(*
:Description: User-facing FB for capturing oversampled metric values and pushing
to tc-otel as compact batched frames.

Lifecycle pattern: declare one FB_Metrics per logical metric, ``Init`` it once
in first cycle, then call ``Observe`` with the value of any IEC scalar (or
STRING / WSTRING) you want to track. The FB:

* Locks the IEC type class on the very first ``Observe`` and rejects later
  calls of a different class — no aggregator-strategy switching mid-flight.
* Optionally rate-limits sampling (``SetSampleIntervalMs``) so a value that
  changes faster than the configured interval is sampled at most once per
  interval. Default 0 = no rate limit (every change is sampled).
* Optionally suppresses redundant samples (``SetChangeDetect``, default TRUE)
  via byte-wise comparison against the last sampled value.
* Buffers samples in an append-only body buffer (8 KB default). On overflow
  the per-frame ``flags.bit1 = ring_overflowed`` is set and additional
  samples are dropped until the next flush.
* Flushes the buffer at the configured push interval (``SetPushIntervalMs``,
  default 1000 ms). Flush also fires from ``Call()`` so users who call
  ``Observe`` only on demand still get punctual pushes.

Each frame carries header + (optional trace context) + name + unit + body.
The body is just ``sample_count * sample_size`` raw bytes — no per-sample
type/length, the receiver knows the layout from the header's ``body_schema``.

Numerics (all signed/unsigned int + REAL + LREAL) widen to LREAL (8 B). BOOL
is one byte. STRING/WSTRING are zero-padded to a per-instance fixed size
configured in ``Init``. Discrete byte-types (BYTE/WORD/DWORD/LWORD/ENUM)
are shipped raw at their native size.

**Example**

.. code-block:: pascal

    VAR
        fbMotorTemp : FB_Metrics;
    END_VAR

    IF _TaskInfo[GETCURTASKINDEXEX()].FirstCycle THEN
        fbMotorTemp.Init('motor.temperature', 'celsius');
        fbMotorTemp.SetSampleIntervalMs(100);   // at most every 100 ms
        fbMotorTemp.SetPushIntervalMs(5000);    // flush every 5 s
    END_IF

    fbMotorTemp.Observe(rTemperature);          // every cycle is fine
    PRG_TaskLog.Call();                         // pumps the per-task sender
*)
{attribute 'reflection'}
FUNCTION_BLOCK FB_Metrics
VAR_INPUT
END_VAR
VAR_OUTPUT
END_VAR
VAR CONSTANT
    (* Each frame is laid out as one contiguous byte array where the header
       grows backward into a 256-byte reserve immediately before the body.
       ADSWRITE reads a single pointer that starts at [HDR_RESERVE - hdrLen]
       and runs through the body — no MEMCPY of either region on flush.

       Header max observed size (v2 frame + 24 B trace_ctx + 63 B name + 15 B
       unit) is ~154 B; 256 B is generous padding. Body is 32 KB per half so
       a true-oversampling DC-timestamp burst (16 B / Numeric slot) fits
       ~2048 samples before mid-window autoflush kicks in. Total per-half =
       HDR_RESERVE + BODY_CAPACITY = 33024 B.

       Autoflush high-water mark: when _nBodyOffset crosses 4/5 of
       BODY_CAPACITY the next append triggers _DoFlush, swapping halves
       mid-window so the burst keeps streaming. *)
    HDR_RESERVE             : UDINT := 256;
    BODY_CAPACITY           : UDINT := 32768;
    BODY_HIGH_WATER         : UDINT := 26214;         // BODY_CAPACITY * 4 / 5
    FRAME_SIZE              : UDINT := 33024;         // HDR_RESERVE + BODY_CAPACITY
END_VAR
VAR
    (* Identification *)
    _bInitialized       : BOOL;
    _sName              : STRING(63);
    _sUnit              : STRING(15);
    _nMetricId          : UDINT;                      // FNV-1a(name)

    (* Type lock — set on first Observe *)
    _eBodySchema        : E_MetricBodySchema;         // eUnknown until first Observe
    _nSampleSize        : UDINT;                      // bytes per sample in body
    _nLockedTypeClass   : __SYSTEM.TYPE_CLASS;
    _nStringSize        : UDINT := 64;                // for eString / eWstring; bytes for eString, chars for eWstring

    (* Phase 8 — A/B frame layout. Each half is one contiguous byte array
       with the header staged into [HDR_RESERVE - hdrLen .. HDR_RESERVE - 1]
       and body samples appended from [HDR_RESERVE..]. Observe writes into
       whichever half is ACTIVE; the pending half stays frozen while the
       sender ships it via ADSWRITE with SRCADDR pointing directly here.
       No MEMCPY of the body on flush. *)
    _aFrameA            : ARRAY[0..33023] OF BYTE;
    _aFrameB            : ARRAY[0..33023] OF BYTE;
    _eActiveBuf         : USINT;                      // 0 = A is active, 1 = B is active

    (* Active-half mutable state. Reset on flush when the active half flips. *)
    _nBodyOffset        : UDINT;                      // bytes appended into active body region (from HDR_RESERVE)
    _nSampleCount       : UDINT;
    _bOverflow          : BOOL;

    (* Pending-half snapshot — owned by the sender from Enqueue until the
       _NotifyFrameSent callback. Stable pointer region:
       frame[HDR_RESERVE - _nPendingHdrLen .. HDR_RESERVE + _nPendingBodyLen - 1]. *)
    _bPending           : BOOL;
    _ePendingBuf        : USINT;                      // 0 = A is pending, 1 = B is pending
    _nPendingHdrLen     : UDINT;
    _nPendingBodyLen    : UDINT;

    (* Change-detect cache — first 64 B of the last sampled value. Long
       strings (>64 B) lose change-detect precision past byte 64; this
       is acceptable for typical state strings. *)
    _abyLastValue       : ARRAY[0..63] OF BYTE;
    _bLastValueValid    : BOOL;
    _bChangeDetect      : BOOL := TRUE;

    (* Timing — uses task cycle counter converted to cycle targets so it
       agrees with FB_TcOtelTaskDiag and survives RtcTime jitter / sync. *)
    _nSampleIntervalMs  : UDINT;                      // 0 = no rate limit
    _nPushIntervalMs    : UDINT := 1000;
    _nLastSampleCycle   : UDINT;
    _bLastSampleSet     : BOOL;
    _nWindowStartCycle  : UDINT;
    _bWindowStartSet    : BOOL;

    (* Window content *)
    _nCycleStart        : UDINT;
    _nCycleEnd          : UDINT;
    _nDcTimeStart       : LINT;
    _nDcTimeEnd         : LINT;
    _bWindowHasSample   : BOOL;

    (* Counters surfaced for online inspection *)
    _nFlushOk           : UDINT;
    _nDropAppend        : UDINT;                      // appends dropped (active body overflow)
    _nDropEmit          : UDINT;                      // sender ring full / ADSWRITE err
    _nDropWindow        : UDINT;                      // window expired while previous still queued
    _nWrongTypeDrops    : UDINT;                      // Observe called with type ≠ locked

    (* Phase 7 — bitmask aggregation. When _nStatMask > 0 and the locked
       schema is numeric, Observe updates the aggregator on every call
       (Welford online for mean/stddev) instead of just rate-limiting.
       At each sample tick popcount(_nStatMask) LREALs are written into
       the body in bit-order (Min, Max, Mean, Sum, Count, StdDev) and the
       aggregator resets. Mask=0 keeps the original raw-sample behaviour. *)
    _nStatMask          : BYTE;                       // E_MetricStat bitmask, 0 = raw
    _nAggSampleSize     : UDINT;                      // popcount(mask) * 8, cached
    _aggMin             : LREAL;
    _aggMax             : LREAL;
    _aggMean            : LREAL;                      // Welford running mean
    _aggSumSq           : LREAL;                      // sum of squared deltas (Welford M2)
    _aggSum             : LREAL;
    _nAggCount          : UDINT;
    _bAggHasSample      : BOOL;                       // first observation in current window seen?

    (* Trace-context binding (Phase 5).
       _pTracer is set persistently by BindTracer — at flush time the
       tracer's innermost open span is snapshotted into the frame.
       _pSpanOverride is set by WithSpan and consumed by the very next
       flush — lets users force a specific span when "innermost" isn't
       what they want. *)
    _pTracer            : REFERENCE TO FB_Trace;
    _pSpanOverride      : REFERENCE TO FB_Span;

    (* Per-sample timestamps (opt-in). When TRUE each body slot is prefixed
       with a 2-byte little-endian u16 cycle offset (relative to
       _nCycleStart). _CheckFlush caps the push window at 0xFFFF cycles to
       keep u16 safe; receiver-side decoders gate on the matching header flag
       METRIC_FLAG_HAS_SAMPLE_TS (0x04). *)
    _bRecordSampleTimes   : BOOL;

    (* High-resolution per-sample timestamps for true oversampling. When TRUE
       each body slot is prefixed with an 8-byte little-endian i64 absolute
       DC time — the raw F_GetActualDcTime64() reading at the Observe call.
       Mutually exclusive with _bRecordSampleTimes; setting both is a
       programming error. Receiver-side decoders gate on the matching header
       flag METRIC_FLAG_HAS_SAMPLE_TS_DC (0x10). Slot stride becomes
       _nSampleSize + 8. No tiebreaker — duplicate DC reads inside one task
       cycle stay duplicate so emitted timestamps don't lie about the
       hardware clock. *)
    _bRecordSampleTimesDc : BOOL;

    (* Phase 2 scope-resolver: instance path of the owning FB.
       FB_Init strips the library + application + variable-name
       segments, leaving (e.g.) ``PRG_Foo.fbBar`` in ``_sLogger``.
       Emitted as the trailing namespace string on the metric
       aggregate frame when non-empty; tc-otel's ScopeResolver
       maps it to the owning FB's TYPE for ``scope.name``. *)
    {attribute 'instance-path'}
    {attribute 'noinit'}
    _sInstancePath      : T_MaxString;
    _sLogger            : T_MaxString;
END_VAR

(*
:Description: Byte pointer to the start of the body region in the ACTIVE frame.

Body writes land at ``_ActiveBodyPtr() + _nBodyOffset``. Swapping buffers
at flush time only toggles ``_eActiveBuf``; subsequent Observe calls land
in the now-fresh half without touching the pending half still being shipped.
*)
METHOD PRIVATE _ActiveBodyPtr : POINTER TO BYTE
IF _eActiveBuf = 0 THEN
    _ActiveBodyPtr := ADR(_aFrameA[HDR_RESERVE]);
ELSE
    _ActiveBodyPtr := ADR(_aFrameB[HDR_RESERVE]);
END_IF
END_METHOD

(*
:Description: Byte pointer to the start of the ACTIVE frame (i.e. the header
reserve base). Used by _DoFlush to position the header immediately before the
body via ``_ActiveFrameAddr() + (HDR_RESERVE - hdrLen)``.
*)
METHOD PRIVATE _ActiveFrameAddr : POINTER TO BYTE
IF _eActiveBuf = 0 THEN
    _ActiveFrameAddr := ADR(_aFrameA[0]);
ELSE
    _ActiveFrameAddr := ADR(_aFrameB[0]);
END_IF
END_METHOD

(*
:Description: Clear the Welford aggregator state at the start of every sample window.
*)
METHOD PRIVATE _AggReset
_aggMin        := 0.0;
_aggMax        := 0.0;
_aggMean       := 0.0;
_aggSumSq      := 0.0;
_aggSum        := 0.0;
_nAggCount     := 0;
_bAggHasSample := FALSE;
END_METHOD

(*
:Description: Fold one observation into the Welford online aggregator.

Maintains running min/max/sum/count exactly, and mean / sum-of-squared-
deltas via Welford so the per-Observe cost stays at ~6 LREAL ops without
ever rebuilding from a stored sample list. StdDev is derived from
``_aggSumSq / (n - 1)`` only at flush time.

Reference: B. P. Welford, *Note on a Method for Calculating Corrected
Sums of Squares and Products*, Technometrics 4(3), 1962.
*)
METHOD PRIVATE _AggUpdate
VAR_INPUT
    fValue : LREAL;
END_VAR
VAR
    fDelta  : LREAL;
    fDelta2 : LREAL;
END_VAR
IF NOT _bAggHasSample THEN
    _aggMin        := fValue;
    _aggMax        := fValue;
    _aggMean       := fValue;
    _aggSumSq      := 0.0;
    _aggSum        := fValue;
    _nAggCount     := 1;
    _bAggHasSample := TRUE;
ELSE
    IF fValue < _aggMin THEN
        _aggMin := fValue;
    END_IF
    IF fValue > _aggMax THEN
        _aggMax := fValue;
    END_IF
    _aggSum    := _aggSum + fValue;
    _nAggCount := _nAggCount + 1;
    fDelta     := fValue - _aggMean;
    _aggMean   := _aggMean + fDelta / UDINT_TO_LREAL(_nAggCount);
    fDelta2    := fValue - _aggMean;
    _aggSumSq  := _aggSumSq + fDelta * fDelta2;
END_IF
END_METHOD

(*
:Description: Widen any IEC numeric (or BOOL) to LREAL.

Returns 0.0 for unsupported types — caller must verify TypeClass first.
Mirrors the dispatch in FB_TcOtelTaskTracer.AddAny so trace and metric
emission see numerics consistently.
*)
METHOD PRIVATE _AnyToLreal : LREAL
VAR_INPUT
    stArg : ANY;
END_VAR
VAR
    pBool  : POINTER TO BYTE;
    pSint  : POINTER TO SINT;
    pInt   : POINTER TO INT;
    pDint  : POINTER TO DINT;
    pLint  : POINTER TO LINT;
    pUsint : POINTER TO USINT;
    pUint  : POINTER TO UINT;
    pUdint : POINTER TO UDINT;
    pUlint : POINTER TO ULINT;
    pReal  : POINTER TO REAL;
    pLreal : POINTER TO LREAL;
END_VAR
CASE stArg.TypeClass OF
    __SYSTEM.TYPE_CLASS.TYPE_BOOL:
        pBool := stArg.pValue;
        IF pBool^ <> 0 THEN
            _AnyToLreal := 1.0;
        ELSE
            _AnyToLreal := 0.0;
        END_IF

    __SYSTEM.TYPE_CLASS.TYPE_SINT:
        pSint := stArg.pValue;
        _AnyToLreal := SINT_TO_LREAL(pSint^);

    __SYSTEM.TYPE_CLASS.TYPE_INT:
        pInt := stArg.pValue;
        _AnyToLreal := INT_TO_LREAL(pInt^);

    __SYSTEM.TYPE_CLASS.TYPE_DINT:
        pDint := stArg.pValue;
        _AnyToLreal := DINT_TO_LREAL(pDint^);

    __SYSTEM.TYPE_CLASS.TYPE_LINT:
        pLint := stArg.pValue;
        _AnyToLreal := LINT_TO_LREAL(pLint^);

    __SYSTEM.TYPE_CLASS.TYPE_USINT,
    __SYSTEM.TYPE_CLASS.TYPE_BYTE:
        pUsint := stArg.pValue;
        _AnyToLreal := USINT_TO_LREAL(pUsint^);

    __SYSTEM.TYPE_CLASS.TYPE_UINT,
    __SYSTEM.TYPE_CLASS.TYPE_WORD:
        pUint := stArg.pValue;
        _AnyToLreal := UINT_TO_LREAL(pUint^);

    __SYSTEM.TYPE_CLASS.TYPE_UDINT,
    __SYSTEM.TYPE_CLASS.TYPE_DWORD:
        pUdint := stArg.pValue;
        _AnyToLreal := UDINT_TO_LREAL(pUdint^);

    __SYSTEM.TYPE_CLASS.TYPE_ULINT,
    __SYSTEM.TYPE_CLASS.TYPE_LWORD:
        pUlint := stArg.pValue;
        _AnyToLreal := ULINT_TO_LREAL(pUlint^);

    __SYSTEM.TYPE_CLASS.TYPE_REAL:
        pReal := stArg.pValue;
        _AnyToLreal := REAL_TO_LREAL(pReal^);

    __SYSTEM.TYPE_CLASS.TYPE_LREAL:
        pLreal := stArg.pValue;
        _AnyToLreal := pLreal^;

    ELSE
        _AnyToLreal := 0.0;
END_CASE
END_METHOD

(*
:Description: Snapshot the current Welford aggregator into the body buffer.

Writes ``popcount(_nStatMask) * 8`` bytes — one LREAL per set bit, in
bit-index order (Min, Max, Mean, Sum, Count, StdDev). Returns FALSE on
body overflow without touching the buffer; the caller marks ``_bOverflow``.

Empty windows (no Observe call landed since the previous snapshot) still
produce a sample slot — all zeros — so ``sample_count`` keeps matching the
expected wall-clock cadence on the receiver side.
*)
METHOD PRIVATE _AppendAggregated : BOOL
VAR_INPUT
    (* Cycle offset for this sample relative to _nCycleStart. Only written
       when _bRecordSampleTimes is TRUE; ignored otherwise. Callers pass 0
       when they don't care. *)
    nCycleOff : UINT;
    (* Absolute DC time for this sample (raw F_GetActualDcTime64). Only
       written when _bRecordSampleTimesDc is TRUE; ignored otherwise. *)
    nDcSample : LINT;
END_VAR
VAR
    pDst    : POINTER TO BYTE;
    nOffset : UDINT;
    nStride : UDINT;
    fStdDev : LREAL;
    fCount  : LREAL;
END_VAR
nStride := _nSampleSize;
IF _bRecordSampleTimes THEN
    nStride := nStride + 2;
ELSIF _bRecordSampleTimesDc THEN
    nStride := nStride + 8;
END_IF
IF (_nBodyOffset + nStride) > BODY_CAPACITY THEN
    _AppendAggregated := FALSE;
    RETURN;
END_IF

pDst    := _ActiveBodyPtr() + _nBodyOffset;
IF _bRecordSampleTimes THEN
    Tc2_System.MEMCPY(pDst, ADR(nCycleOff), 2);
    pDst := pDst + 2;
ELSIF _bRecordSampleTimesDc THEN
    Tc2_System.MEMCPY(pDst, ADR(nDcSample), 8);
    pDst := pDst + 8;
END_IF
nOffset := 0;

IF (_nStatMask AND E_MetricStat.eMin) <> 0 THEN
    Tc2_System.MEMCPY(pDst + nOffset, ADR(_aggMin), 8);
    nOffset := nOffset + 8;
END_IF
IF (_nStatMask AND E_MetricStat.eMax) <> 0 THEN
    Tc2_System.MEMCPY(pDst + nOffset, ADR(_aggMax), 8);
    nOffset := nOffset + 8;
END_IF
IF (_nStatMask AND E_MetricStat.eMean) <> 0 THEN
    Tc2_System.MEMCPY(pDst + nOffset, ADR(_aggMean), 8);
    nOffset := nOffset + 8;
END_IF
IF (_nStatMask AND E_MetricStat.eSum) <> 0 THEN
    Tc2_System.MEMCPY(pDst + nOffset, ADR(_aggSum), 8);
    nOffset := nOffset + 8;
END_IF
IF (_nStatMask AND E_MetricStat.eCount) <> 0 THEN
    fCount := UDINT_TO_LREAL(_nAggCount);
    Tc2_System.MEMCPY(pDst + nOffset, ADR(fCount), 8);
    nOffset := nOffset + 8;
END_IF
IF (_nStatMask AND E_MetricStat.eStdDev) <> 0 THEN
    IF _nAggCount > 1 THEN
        fStdDev := SQRT(_aggSumSq / UDINT_TO_LREAL(_nAggCount - 1));
    ELSE
        fStdDev := 0.0;
    END_IF
    Tc2_System.MEMCPY(pDst + nOffset, ADR(fStdDev), 8);
    nOffset := nOffset + 8;
END_IF

_nBodyOffset      := _nBodyOffset + nStride;
_nSampleCount     := _nSampleCount + 1;
_AppendAggregated := TRUE;
END_METHOD

(*
:Description: Write one sample of the locked schema into the body buffer.

Returns FALSE when the body is full — caller sets ``_bOverflow``.
*)
METHOD PRIVATE _AppendSample : BOOL
VAR_INPUT
    stArg     : ANY;
    (* Cycle offset for this sample relative to _nCycleStart. Only written
       when _bRecordSampleTimes is TRUE; ignored otherwise. Callers pass 0
       when they don't care. *)
    nCycleOff : UINT;
    (* Absolute DC time for this sample (raw F_GetActualDcTime64). Only
       written when _bRecordSampleTimesDc is TRUE; ignored otherwise. *)
    nDcSample : LINT;
END_VAR
VAR
    fLreal     : LREAL;
    nStrLen    : UDINT;
    nCopyLen   : UDINT;
    nStride    : UDINT;
    pDst       : POINTER TO BYTE;
    pWstr      : POINTER TO WSTRING(255);
END_VAR
nStride := _nSampleSize;
IF _bRecordSampleTimes THEN
    nStride := nStride + 2;
ELSIF _bRecordSampleTimesDc THEN
    nStride := nStride + 8;
END_IF
IF (_nBodyOffset + nStride) > BODY_CAPACITY THEN
    _AppendSample := FALSE;
    RETURN;
END_IF

pDst := _ActiveBodyPtr() + _nBodyOffset;
IF _bRecordSampleTimes THEN
    Tc2_System.MEMCPY(pDst, ADR(nCycleOff), 2);
    pDst := pDst + 2;
ELSIF _bRecordSampleTimesDc THEN
    Tc2_System.MEMCPY(pDst, ADR(nDcSample), 8);
    pDst := pDst + 8;
END_IF

CASE _eBodySchema OF
    E_MetricBodySchema.eBool:
        IF Tc2_Utilities.PBYTE_TO_BYTE(stArg.pValue) <> 0 THEN
            pDst^ := 1;
        ELSE
            pDst^ := 0;
        END_IF

    E_MetricBodySchema.eNumeric:
        fLreal := _AnyToLreal(stArg);
        Tc2_System.MEMCPY(pDst, ADR(fLreal), 8);

    E_MetricBodySchema.eDiscrete:
        nCopyLen := DINT_TO_UDINT(stArg.diSize);
        IF nCopyLen > _nSampleSize THEN
            nCopyLen := _nSampleSize;
        END_IF
        Tc2_System.MEMCPY(pDst, stArg.pValue, nCopyLen);
        IF nCopyLen < _nSampleSize THEN
            Tc2_System.MEMSET(pDst + nCopyLen, 0, _nSampleSize - nCopyLen);
        END_IF

    E_MetricBodySchema.eString:
        Tc2_System.MEMSET(pDst, 0, _nSampleSize);
        nStrLen := Tc2_Utilities.LEN2(stArg.pValue);
        IF nStrLen > _nSampleSize THEN
            nStrLen := _nSampleSize;
        END_IF
        IF nStrLen > 0 THEN
            Tc2_System.MEMCPY(pDst, stArg.pValue, nStrLen);
        END_IF

    E_MetricBodySchema.eWstring:
        Tc2_System.MEMSET(pDst, 0, _nSampleSize);
        (* WLEN returns characters; we ship 2 B each, capped at _nSampleSize bytes.
           Typed-pointer cast first because WLEN can't take PVOID directly —
           same pattern FB_LogEntry._WriteWString uses. *)
        pWstr := stArg.pValue;
        nStrLen := INT_TO_UDINT(Tc2_Standard.WLEN(pWstr^)) * 2;
        IF nStrLen > _nSampleSize THEN
            nStrLen := _nSampleSize;
        END_IF
        IF nStrLen > 0 THEN
            Tc2_System.MEMCPY(pDst, stArg.pValue, nStrLen);
        END_IF

    ELSE
        _AppendSample := FALSE;
        RETURN;
END_CASE

_nBodyOffset  := _nBodyOffset + nStride;
_nSampleCount := _nSampleCount + 1;

_AppendSample := TRUE;
END_METHOD

(*
:Description: Flush if push window has elapsed.

Window timing is cycle-based (mirrors ``FB_TcOtelTaskDiag.CheckFlush``):
``target_cycles = push_interval_ms * 1000 / cycle_time_us``. Doesn't fire
when the buffer is empty — empty windows just slide the start cycle
forward.
*)
METHOD PRIVATE _CheckFlush
VAR
    nTaskIdx       : DINT;
    pTi            : POINTER TO PlcTaskSystemInfo;
    nNowCycle      : UDINT;
    nCycleTimeUs   : UDINT;
    nTargetCycles  : UDINT;
END_VAR
nTaskIdx := Tc2_Utilities.GETCURTASKINDEXEX();
IF nTaskIdx <= 0 THEN
    RETURN;
END_IF
pTi := ADR(TwinCAT_SystemInfoVarList._TaskInfo[nTaskIdx]);

nCycleTimeUs := pTi^.CycleTime / 10;
IF nCycleTimeUs = 0 THEN
    nCycleTimeUs := 1000; (* fallback: assume 1 ms *)
END_IF
nTargetCycles := (_nPushIntervalMs * 1000) / nCycleTimeUs;
IF nTargetCycles = 0 THEN
    nTargetCycles := 1;
END_IF

(* When per-sample timestamps are active, cap the window at the u16 ceiling
   so the per-sample cycle-offset never overflows. Observable effect: an
   earlier autoflush for extreme configs (e.g. 20 s push window on a 250 µs
   task). WithSpan pins may be consumed by the autoflush rather than the
   natural flush — use BindTracer for spans that outlive one window. *)
IF _bRecordSampleTimes AND nTargetCycles > 16#FFFF THEN
    nTargetCycles := 16#FFFF;
END_IF

nNowCycle := pTi^.CycleCount;
IF NOT _bWindowStartSet OR nNowCycle < _nWindowStartCycle THEN
    _nWindowStartCycle := nNowCycle;
    _bWindowStartSet   := TRUE;
    RETURN;
END_IF

IF (nNowCycle - _nWindowStartCycle) < nTargetCycles THEN
    RETURN;
END_IF

IF _nSampleCount > 0 THEN
    _DoFlush();
END_IF
_nWindowStartCycle := nNowCycle;
END_METHOD

(*
:Description: Finalize the active window into a sendable frame and enqueue for the sender.

Phase 8 — zero-copy queued dispatch:

1. If the previous window is still queued (``_bPending``) the sender has
   fallen behind. Increment ``_nDropWindow`` and reset the active half —
   we cannot touch the pending half nor duplicate ourselves in the queue.
2. Otherwise: build the header into a small stack staging (≤ ~160 B),
   MEMCPY the staged header into the active frame's reserve region so it
   sits directly before the body (one contiguous byte run), snapshot the
   pending metadata (buf index, hdr len, body len), flip ``_eActiveBuf``,
   reset the now-active (previously empty) half, and call
   ``sender.Enqueue(THIS)``.

The sender later calls ``_GetPendingPtr`` / ``_GetPendingLen`` to read the
frame pointer + length directly into ADSWRITE, and ``_NotifyFrameSent``
when the transfer completes. The body buffer is never MEMCPY'd.
*)
METHOD PRIVATE _DoFlush
VAR
    stHeader    : ST_PushMetricAggHeader;
    abyHdr      : ARRAY[0..255] OF BYTE;   // header(52) + trace(24) + name(63) + unit(15) + ns_len(1) + ns(127) ≤ 282
    nHdrLen     : UDINT;
    nNameLen    : UDINT;
    nUnitLen    : UDINT;
    nNsLen      : UDINT;
    byNsLen     : BYTE;
    refSender   : REFERENCE TO FB_TcOtelTaskMetrics;
    refSpan     : REFERENCE TO FB_Span;
    pActiveBase : POINTER TO BYTE;
END_VAR
(* Backlog guard: if the sender is still shipping our previous frame, the
   pending half is in use and we have no clean buffer to swap into. Drop
   this window rather than risk body corruption. In practice this only
   fires during a dead / slow tc-otel endpoint. *)
IF _bPending THEN
    _nDropWindow      := _nDropWindow + 1;
    _nBodyOffset      := 0;
    _nSampleCount     := 0;
    _bOverflow        := FALSE;
    _bWindowHasSample := FALSE;
    _nCycleStart      := 0;
    _nCycleEnd        := 0;
    _nDcTimeStart     := 0;
    _nDcTimeEnd       := 0;
    RETURN;
END_IF

(* Resolve trace context: per-flush WithSpan override beats persistent
   BindTracer. Both candidates and the chosen handle stay as REFERENCE TO —
   nullable via REF= 0 + __ISVALIDREF, no pointer round-trip needed. *)
refSpan REF= 0;
IF __ISVALIDREF(_pSpanOverride) THEN
    refSpan REF= _pSpanOverride;
ELSIF __ISVALIDREF(_pTracer) THEN
    refSpan REF= _pTracer.InnermostSpan;
END_IF

(* Build fixed header. *)
stHeader.nVersion         := 2;
stHeader.nEventType       := 21;
stHeader.nFlags           := 0;
IF _bOverflow THEN
    stHeader.nFlags := stHeader.nFlags OR 16#02;    (* bit1 = ring_overflowed *)
END_IF
IF __ISVALIDREF(refSpan) THEN
    stHeader.nFlags := stHeader.nFlags OR 16#01;    (* bit0 = has_trace_ctx *)
END_IF
IF _bRecordSampleTimes THEN
    stHeader.nFlags := stHeader.nFlags OR 16#04;    (* bit2 = has_sample_ts *)
END_IF
IF _bRecordSampleTimesDc THEN
    stHeader.nFlags := stHeader.nFlags OR 16#10;    (* bit4 = has_sample_ts_dc *)
END_IF
nNsLen := Tc2_Utilities.LEN2(ADR(_sLogger));
IF nNsLen > 127 THEN
    nNsLen := 127;
END_IF
IF nNsLen > 0 THEN
    stHeader.nFlags := stHeader.nFlags OR 16#08;    (* bit3 = has_namespace *)
END_IF
stHeader.eBodySchema      := _eBodySchema;
stHeader.nSampleSize      := _nSampleSize;
stHeader.nSampleCount     := _nSampleCount;
stHeader.nMetricId        := _nMetricId;
stHeader.nTaskIndex       := TO_USINT(Tc2_Utilities.GETCURTASKINDEXEX());
stHeader.nStatMask        := _nStatMask;
stHeader.nCycleCountStart := _nCycleStart;
stHeader.nCycleCountEnd   := _nCycleEnd;
stHeader.nDcTimeStart     := _nDcTimeStart;
stHeader.nDcTimeEnd       := _nDcTimeEnd;

nNameLen := Tc2_Utilities.LEN2(ADR(_sName));
IF nNameLen > 63 THEN
    nNameLen := 63;
END_IF
nUnitLen := Tc2_Utilities.LEN2(ADR(_sUnit));
IF nUnitLen > 15 THEN
    nUnitLen := 15;
END_IF
stHeader.nNameLen := TO_BYTE(nNameLen);
stHeader.nUnitLen := TO_BYTE(nUnitLen);

(* Stage [header | (trace_ctx) | name | unit] on the stack. *)
Tc2_System.MEMCPY(ADR(abyHdr), ADR(stHeader), SIZEOF(stHeader));
nHdrLen := SIZEOF(stHeader);

IF __ISVALIDREF(refSpan) THEN
    Tc2_System.MEMCPY(ADR(abyHdr) + nHdrLen,      ADR(refSpan._abTraceId[0]), 16);
    Tc2_System.MEMCPY(ADR(abyHdr) + nHdrLen + 16, ADR(refSpan._abSpanId[0]),  8);
    nHdrLen := nHdrLen + 24;
END_IF

(* Consume per-flush span override — BindTracer stays, WithSpan is one-shot. *)
_pSpanOverride REF= 0;

IF nNameLen > 0 THEN
    Tc2_System.MEMCPY(ADR(abyHdr) + nHdrLen, ADR(_sName), nNameLen);
    nHdrLen := nHdrLen + nNameLen;
END_IF
IF nUnitLen > 0 THEN
    Tc2_System.MEMCPY(ADR(abyHdr) + nHdrLen, ADR(_sUnit), nUnitLen);
    nHdrLen := nHdrLen + nUnitLen;
END_IF
IF nNsLen > 0 THEN
    (* Phase 2 scope-resolver: ns_len(1) + namespace(ns_len). *)
    byNsLen := TO_BYTE(nNsLen);
    Tc2_System.MEMCPY(ADR(abyHdr) + nHdrLen,     ADR(byNsLen),   1);
    Tc2_System.MEMCPY(ADR(abyHdr) + nHdrLen + 1, ADR(_sLogger),  nNsLen);
    nHdrLen := nHdrLen + 1 + nNsLen;
END_IF

(* Defensive clamp: the header reserve is HDR_RESERVE bytes. Oversized
   headers would overlap the body. In practice nHdrLen ≤ 154. *)
IF nHdrLen > HDR_RESERVE THEN
    _nDropEmit := _nDropEmit + 1;
    (* Reset window and bail — don't corrupt the frame layout. *)
    _nBodyOffset      := 0;
    _nSampleCount     := 0;
    _bOverflow        := FALSE;
    _bWindowHasSample := FALSE;
    _nCycleStart      := 0;
    _nCycleEnd        := 0;
    _nDcTimeStart     := 0;
    _nDcTimeEnd       := 0;
    RETURN;
END_IF

(* Position the staged header so its last byte sits at offset HDR_RESERVE-1
   of the active frame — i.e. flush against the body start. Single MEMCPY
   of ≤ 160 B; no body copy. *)
pActiveBase := _ActiveFrameAddr();
Tc2_System.MEMCPY(pActiveBase + (HDR_RESERVE - nHdrLen), ADR(abyHdr), nHdrLen);

(* Snapshot pending metadata: the active (now-to-be-shipped) half. *)
_ePendingBuf     := _eActiveBuf;
_nPendingHdrLen  := nHdrLen;
_nPendingBodyLen := _nBodyOffset;
_bPending        := TRUE;

(* Flip active → the other half. Reset the new-active mutable state. *)
IF _eActiveBuf = 0 THEN
    _eActiveBuf := 1;
ELSE
    _eActiveBuf := 0;
END_IF
_nBodyOffset      := 0;
_nSampleCount     := 0;
_bOverflow        := FALSE;
_bWindowHasSample := FALSE;
_nCycleStart      := 0;
_nCycleEnd        := 0;
_nDcTimeStart     := 0;
_nDcTimeEnd       := 0;

(* Hand the pending half to the sender's dispatch ring. *)
refSender REF= PRG_TaskLog.TaskMetrics;
IF __ISVALIDREF(refSender) THEN
    IF NOT refSender.Enqueue(THIS) THEN
        (* Ring overflow — real drop. Release the pending half so the next
           window can still flush, and count as emit drop. *)
        _bPending  := FALSE;
        _nDropEmit := _nDropEmit + 1;
    END_IF
ELSE
    (* Sender missing — treat like ring overflow. *)
    _bPending  := FALSE;
    _nDropEmit := _nDropEmit + 1;
END_IF
END_METHOD

(*
:Description: INTERNAL — total bytes of the frame currently in the sender queue.

Called by ``FB_TcOtelTaskMetrics._KickHead`` to populate ADSWRITE.LEN.
Returns 0 when ``_bPending`` is FALSE (spurious call — sender should ignore).
*)
METHOD INTERNAL _GetPendingLen : UDINT
IF _bPending THEN
    _GetPendingLen := _nPendingHdrLen + _nPendingBodyLen;
ELSE
    _GetPendingLen := 0;
END_IF
END_METHOD

(*
:Description: INTERNAL — byte pointer to the first byte of the pending frame.

Frame layout in the pending half (``_ePendingBuf``):
  [HDR_RESERVE - _nPendingHdrLen .. HDR_RESERVE - 1]  header + trace + name + unit
  [HDR_RESERVE .. HDR_RESERVE + _nPendingBodyLen - 1] body samples
So the frame starts at ``frame[HDR_RESERVE - _nPendingHdrLen]`` and runs
``_nPendingHdrLen + _nPendingBodyLen`` bytes — a single contiguous ADS range.

Called by ``FB_TcOtelTaskMetrics._KickHead`` to populate ADSWRITE.SRCADDR.
Returns 0 when no frame is pending.
*)
METHOD INTERNAL _GetPendingPtr : PVOID
IF NOT _bPending THEN
    _GetPendingPtr := 0;
    RETURN;
END_IF

IF _ePendingBuf = 0 THEN
    _GetPendingPtr := ADR(_aFrameA[0]) + (HDR_RESERVE - _nPendingHdrLen);
ELSE
    _GetPendingPtr := ADR(_aFrameB[0]) + (HDR_RESERVE - _nPendingHdrLen);
END_IF
END_METHOD

(*
:Description: Map the IEC type class of the first Observe call to a body schema.

Returns FALSE for unsupported types (TIME, DATE, structures, arrays, etc.)
so Observe can drop those gracefully and surface via _nWrongTypeDrops.
*)
METHOD PRIVATE _LockSchema : BOOL
VAR_INPUT
    stArg : ANY;
END_VAR
CASE stArg.TypeClass OF
    __SYSTEM.TYPE_CLASS.TYPE_BOOL:
        _eBodySchema := E_MetricBodySchema.eBool;
        _nSampleSize := 1;

    __SYSTEM.TYPE_CLASS.TYPE_SINT,
    __SYSTEM.TYPE_CLASS.TYPE_INT,
    __SYSTEM.TYPE_CLASS.TYPE_DINT,
    __SYSTEM.TYPE_CLASS.TYPE_LINT,
    __SYSTEM.TYPE_CLASS.TYPE_USINT,
    __SYSTEM.TYPE_CLASS.TYPE_UINT,
    __SYSTEM.TYPE_CLASS.TYPE_UDINT,
    __SYSTEM.TYPE_CLASS.TYPE_ULINT,
    __SYSTEM.TYPE_CLASS.TYPE_REAL,
    __SYSTEM.TYPE_CLASS.TYPE_LREAL:
        IF _nStatMask <> 0 THEN
            _eBodySchema := E_MetricBodySchema.eNumericAggregated;
            _nSampleSize := _nAggSampleSize;
        ELSE
            _eBodySchema := E_MetricBodySchema.eNumeric;
            _nSampleSize := 8;     (* widened to LREAL *)
        END_IF

    __SYSTEM.TYPE_CLASS.TYPE_BYTE,
    __SYSTEM.TYPE_CLASS.TYPE_WORD,
    __SYSTEM.TYPE_CLASS.TYPE_DWORD,
    __SYSTEM.TYPE_CLASS.TYPE_LWORD,
    __SYSTEM.TYPE_CLASS.TYPE_ENUM:
        _eBodySchema := E_MetricBodySchema.eDiscrete;
        _nSampleSize := DINT_TO_UDINT(stArg.diSize);

    __SYSTEM.TYPE_CLASS.TYPE_STRING:
        _eBodySchema := E_MetricBodySchema.eString;
        _nSampleSize := _nStringSize;
        F_InternalLog(
            E_LogLevel.eWarn,
            'FB_Metrics._LockSchema',
            'Unsupported TypeClass=%d for metric %s',
            Tc2_Utilities.F_UDINT(stArg.TypeClass),
            Tc2_Utilities.F_StringEx(_sName),
            Tc2_Utilities.EMPTY_ARG_VALUE,
            Tc2_Utilities.EMPTY_ARG_VALUE
        );
        _LockSchema := FALSE;
        RETURN;

    __SYSTEM.TYPE_CLASS.TYPE_WSTRING:
        _eBodySchema := E_MetricBodySchema.eWstring;
        _nSampleSize := _nStringSize * 2;
        F_InternalLog(
            E_LogLevel.eWarn,
            'FB_Metrics._LockSchema',
            'Unsupported TypeClass=%d for metric %s',
            Tc2_Utilities.F_UDINT(stArg.TypeClass),
            Tc2_Utilities.F_StringEx(_sName),
            Tc2_Utilities.EMPTY_ARG_VALUE,
            Tc2_Utilities.EMPTY_ARG_VALUE
        );
        _LockSchema := FALSE;
        RETURN;

    ELSE
        F_InternalLog(
            E_LogLevel.eWarn,
            'FB_Metrics._LockSchema',
            'Unsupported TypeClass=%d for metric %s',
            Tc2_Utilities.F_UDINT(stArg.TypeClass),
            Tc2_Utilities.F_StringEx(_sName),
            Tc2_Utilities.EMPTY_ARG_VALUE,
            Tc2_Utilities.EMPTY_ARG_VALUE
        );
        _LockSchema := FALSE;
        RETURN;
END_CASE

_nLockedTypeClass := stArg.TypeClass;
_LockSchema       := TRUE;
END_METHOD

(*
:Description: INTERNAL — sender completion callback.

Called by ``FB_TcOtelTaskMetrics.Call`` once ADSWRITE finishes (success, ADS
error, or watchdog). Releases the pending half so the next ``_DoFlush`` can
swap into it, and updates per-metric counters.

Do not call from user code.
*)
METHOD INTERNAL _NotifyFrameSent
VAR_INPUT
    bOk : BOOL;
END_VAR
IF bOk THEN
    _nFlushOk := _nFlushOk + 1;
ELSE
    _nDropEmit := _nDropEmit + 1;
END_IF

_bPending        := FALSE;
_nPendingHdrLen  := 0;
_nPendingBodyLen := 0;
END_METHOD

(*
:Description: Live DC time, falling back to cycle-start task DC time.

Same fallback as FB_TcOtelTaskTracer._NowDcTime — keeps metric and trace
timestamps comparable.
*)
METHOD PRIVATE _NowDcTime : LINT
VAR
    nTaskIdx : DINT;
END_VAR
_NowDcTime := TO_LINT(Tc2_EtherCAT.F_GetActualDcTime64());
IF _NowDcTime = 0 THEN
    nTaskIdx := Tc2_Utilities.GETCURTASKINDEXEX();
    IF nTaskIdx > 0 THEN
        _NowDcTime := TwinCAT_SystemInfoVarList._TaskInfo[nTaskIdx].DcTaskTime;
    END_IF
END_IF
END_METHOD

(*
:Description: Bit-count of a BYTE — used to size the aggregated sample.

Trivial loop is fine for an 8-bit value; called once per SetAggregation,
not per cycle.
*)
METHOD PRIVATE _PopCount8 : UDINT
VAR_INPUT
    nByte : BYTE;
END_VAR
VAR
    nBit : INT;
END_VAR
_PopCount8 := 0;
FOR nBit := 0 TO 7 DO
    IF (nByte AND SHL(BYTE#1, nBit)) <> 0 THEN
        _PopCount8 := _PopCount8 + 1;
    END_IF
END_FOR
END_METHOD

(*
:Description: Bind this metric to an FB_TcOtelTracer for trace exemplar correlation.

Read-at-flush-time semantic: every ``_DoFlush`` snapshots the tracer's
**currently** innermost-open span (trace_id + span_id) into the wire
header. The span's ID gets promoted to an OTel Exemplar on every data
point in that batch so Grafana / Tempo render "View trace" links.

What ends up on the frame:

* a span is open on the bound tracer at flush time → that span's trace_id
* no span open (all ``End``'d, or never ``Begin``'d) → no trace bytes, frame is 24 B shorter
* ``BindTracer(0)`` → no trace bytes

A span that opens **and** closes between two flushes leaves no trace on
either frame — if that matters, use ``WithSpan`` or call ``Flush``
before ``End``.

Pass ``0`` to unbind. Idempotent — safe to call repeatedly.

**Example**

.. code-block:: pascal

    VAR
        _tracer : FB_TcOtelTracer;
        _temp   : FB_Metrics;
    END_VAR

    IF _TaskInfo[GETCURTASKINDEXEX()].FirstCycle THEN
        _temp.Init('motor.temperature', 'celsius');
        _temp.BindTracer(_tracer);
    END_IF
*)
METHOD PUBLIC BindTracer : BOOL
VAR_INPUT
    pTracer : REFERENCE TO FB_Trace;
END_VAR
_pTracer REF= pTracer;
BindTracer := TRUE;
END_METHOD

(*
:Description: Drives push-window check.

Only needed when the user calls ``Observe`` sporadically (so a long quiet
period would otherwise delay flush past its window). When ``Observe`` is
called every cycle this is redundant but harmless.
*)
METHOD PUBLIC Call
IF _bInitialized THEN
    _CheckFlush();
END_IF
END_METHOD

(*
:Description: Flush any buffered samples before this FB instance is destroyed.

Online change / program stop / FB deletion all route through here — without
this, the last partial window would be silently lost.
*)
METHOD FB_exit : BOOL
VAR_INPUT
    bInCopyCode : BOOL;
END_VAR
(* Cold Reset / RT shutdown destroys FB instances in undefined order.
   PRG_TaskLog.TaskMetrics may be torn down before us; calling
   Dequeue on a dangling reference segfaults inside the AuxTask
   (__ISVALIDREF catches NULL only, not dangling-after-free). Buffered
   samples on shutdown are lost — acceptable, no consumer remains
   after the Reset.

   Online change (bInCopyCode = TRUE) preserves both old and new
   instances in memory; flushing here would double-emit if the new
   instance also flushes. *)
FB_exit := TRUE;
END_METHOD

// Phase 2 scope-resolver: derive _sLogger from the FB's instance
// path. Strips library + application + variable-name segments,
// leaving (e.g.) ``PRG_TestSimpleApi.fbMotor`` so the OTel
// ScopeResolver maps the frame to the OWNING FB's type for
// ``InstrumentationScope.name``. Mirrors FB_Log.FB_Init.
METHOD FB_Init: BOOL
VAR_INPUT
    bInitRetains: BOOL;
    bInCopyCode: BOOL;
END_VAR
VAR
    nFindIdx : INT;
    i        : INT;
    nLastDot : INT;
END_VAR
nFindIdx := Tc2_Standard.FIND(_sInstancePath, '.');
IF nFindIdx > 0 THEN
    _sInstancePath := Tc2_Standard.DELETE(_sInstancePath, nFindIdx + 1, 0);
    nFindIdx := Tc2_Standard.FIND(_sInstancePath, '.');
    IF nFindIdx > 0 THEN
        _sInstancePath := Tc2_Standard.DELETE(_sInstancePath, nFindIdx + 1, 0);
        nLastDot := 0;
        FOR i := Tc2_Standard.LEN(_sInstancePath) TO 1 BY -1 DO
            IF Tc2_Standard.MID(_sInstancePath, 1, i) = '.' THEN
                nLastDot := i;
                EXIT;
            END_IF
        END_FOR
        IF nLastDot > 1 THEN
            _sLogger := Tc2_Standard.LEFT(_sInstancePath, nLastDot - 1);
        ELSE
            _sLogger := _sInstancePath;
        END_IF
    END_IF
END_IF

FB_Init := TRUE;
END_METHOD

(*
:Description: Force-flush the buffered samples now, regardless of push window.

No-op when the buffer is empty.
*)
METHOD PUBLIC Flush : BOOL
IF _bInitialized AND _nSampleCount > 0 THEN
    _DoFlush();
END_IF
Flush := TRUE;
END_METHOD

(*
:Description: One-time configuration of the metric identity.

Idempotent — recomputes the FNV-1a metric id from the current name. Safe
to call from FirstCycle. ``nStringSize`` is only meaningful when the
locked schema turns out to be eString / eWstring; ignored for numerics.
*)
METHOD PUBLIC Init : BOOL
VAR_INPUT
    sName       : STRING(63);
    sUnit       : STRING(15) := '';
    nStringSize : UDINT      := 64;       // bytes per string sample (chars for WSTRING)
END_VAR
VAR
    i      : INT;
    nLen   : INT;
    nHash  : UDINT;
    pBytes : POINTER TO BYTE;
END_VAR
_sName       := sName;
_sUnit       := sUnit;
_nStringSize := nStringSize;
IF _nStringSize = 0 THEN
    _nStringSize := 64;
END_IF
IF _nStringSize > 255 THEN
    _nStringSize := 255;
END_IF

(* FNV-1a 32-bit over the name bytes. Stable across runs as long as the
   name string doesn't change. *)
nHash := UDINT#16#811C9DC5;
nLen  := Tc2_Standard.LEN(_sName);
IF nLen > 0 THEN
    pBytes := ADR(_sName);
    FOR i := 0 TO nLen - 1 DO
        nHash := (nHash XOR BYTE_TO_UDINT(pBytes[i])) * UDINT#16#01000193;
    END_FOR
END_IF
_nMetricId    := nHash;

_bInitialized := TRUE;
Init          := TRUE;
END_METHOD

PROPERTY PUBLIC MetricId : UDINT
GET
MetricId := _nMetricId;
END_GET
END_PROPERTY

(*
:Description: Capture one observation of the metric value.

Returns FALSE only on hard errors (Init not called, unsupported type on
first call, type changed after lock). Successful sample-suppression by
rate-limit or change-detect still returns TRUE — the FB did its job by
deciding the value didn't need to be stored.

Safe to call every cycle — internal rate-limit makes that cheap.
*)
METHOD PUBLIC Observe : BOOL
VAR_INPUT
    stArg : ANY;
END_VAR
VAR
    nTaskIdx       : DINT;
    pTi            : POINTER TO PlcTaskSystemInfo;
    nNowCycle      : UDINT;
    nCycleTimeUs   : UDINT;
    nSampleTargetCycles : UDINT;
    nCmpLen        : UDINT;
    nDcNow         : LINT;
    fLrealForAgg   : LREAL;     // widened sample for the online aggregator
    bAggMode       : BOOL;      // shorthand for "stat-mask aggregation active"
    nCycleOff      : UINT;      // per-sample offset for optional sample-TS
END_VAR
IF NOT _bInitialized OR stArg.pValue = 0 THEN
    Observe := FALSE;
    RETURN;
END_IF

IF _eBodySchema = E_MetricBodySchema.eString OR _eBodySchema = E_MetricBodySchema.eWstring THEN
	_nWrongTypeDrops := _nWrongTypeDrops + 1;
	Observe := FALSE;
	RETURN;
END_IF

(* Lock schema on first call. *)
IF _eBodySchema = E_MetricBodySchema.eUnknown THEN
    IF NOT _LockSchema(stArg) THEN
        _nWrongTypeDrops := _nWrongTypeDrops + 1;
        Observe := FALSE;
        RETURN;
    END_IF
ELSIF _nLockedTypeClass <> stArg.TypeClass THEN
    F_InternalLog(
        E_LogLevel.eWarn,
        'FB_Metrics.Observe',
        'TypeClass mismatch for %s (locked=%d got=%d)',
        Tc2_Utilities.F_StringEx(_sName),
        Tc2_Utilities.F_UDINT(_nLockedTypeClass),
        Tc2_Utilities.F_UDINT(stArg.TypeClass),
        Tc2_Utilities.EMPTY_ARG_VALUE
    );
    _nWrongTypeDrops := _nWrongTypeDrops + 1;
    Observe := FALSE;
    RETURN;
END_IF

nTaskIdx := Tc2_Utilities.GETCURTASKINDEXEX();
IF nTaskIdx <= 0 THEN
    Observe := FALSE;
    RETURN;
END_IF
pTi := ADR(TwinCAT_SystemInfoVarList._TaskInfo[nTaskIdx]);
nNowCycle := pTi^.CycleCount;

bAggMode := _eBodySchema = E_MetricBodySchema.eNumericAggregated;

(* Aggregation: in eNumericAggregated mode the aggregator absorbs every
   single Observe call (Welford online for mean/stddev). The rate-limit
   below still gates how often we *snapshot* the aggregator into the body
   buffer — but no value is dropped between ticks. *)
IF bAggMode THEN
    fLrealForAgg := _AnyToLreal(stArg);
    _AggUpdate(fLrealForAgg);
END_IF

(* Sample-interval rate limit (cycle-based, derived from CycleTime). *)
IF _nSampleIntervalMs > 0 AND _bLastSampleSet THEN
    nCycleTimeUs := pTi^.CycleTime / 10;
    IF nCycleTimeUs = 0 THEN
        nCycleTimeUs := 1000;
    END_IF
    nSampleTargetCycles := (_nSampleIntervalMs * 1000) / nCycleTimeUs;
    IF nSampleTargetCycles = 0 THEN
        nSampleTargetCycles := 1;
    END_IF
    IF (nNowCycle - _nLastSampleCycle) < nSampleTargetCycles THEN
        Observe := TRUE;
        RETURN;
    END_IF
END_IF

(* Change-detect path (raw mode only — for aggregated mode every Observe
   already updated the aggregator above, no point in suppressing). *)
IF NOT bAggMode AND _bChangeDetect AND _bLastValueValid THEN
    nCmpLen := _nSampleSize;
    IF nCmpLen > SIZEOF(_abyLastValue) THEN
        nCmpLen := SIZEOF(_abyLastValue);
    END_IF
    IF Tc2_System.MEMCMP(stArg.pValue, ADR(_abyLastValue), nCmpLen) = 0 THEN
        (* Even on no-change we still update last-sample timestamp so the
           rate-limit window resets — so a value that resumes changing right
           after the interval doesn't have to wait an extra slot. *)
        _nLastSampleCycle := nNowCycle;
        _bLastSampleSet   := TRUE;
        Observe := TRUE;
        RETURN;
    END_IF
END_IF

(* Window timing must be established BEFORE the append so the per-sample
   cycle offset is well-defined on the very first sample. Moving this block
   up changes no observable semantics in the default path — _nCycleStart /
   _nDcTimeStart were overwritten by this sample anyway — but guarantees
   that _bRecordSampleTimes sees a valid reference point. *)
nDcNow := _NowDcTime();
IF NOT _bWindowHasSample THEN
    _nCycleStart      := nNowCycle;
    _nDcTimeStart     := nDcNow;
    _bWindowHasSample := TRUE;
END_IF
_nCycleEnd   := nNowCycle;
_nDcTimeEnd  := nDcNow;

(* u16 offset: safe because _CheckFlush caps the window at 0xFFFF cycles
   whenever _bRecordSampleTimes is active. When the flag is off, the value
   is unused but we still clamp defensively. *)
IF (nNowCycle - _nCycleStart) > 16#FFFF THEN
    nCycleOff := 16#FFFF;
ELSE
    nCycleOff := TO_UINT(nNowCycle - _nCycleStart);
END_IF

IF bAggMode THEN
    (* Snapshot the aggregator into the body, then reset for the next window.
       _AppendAggregated falls through to FALSE only on body overflow — bail
       early in that case, the old aggregator state would be wrong to keep
       around for the next snapshot anyway. *)
    IF NOT _AppendAggregated(nCycleOff, nDcNow) THEN
        _bOverflow   := TRUE;
        _nDropAppend := _nDropAppend + 1;
    END_IF
    _AggReset();
ELSE
    (* Raw append (single value per sample tick). *)
    IF NOT _AppendSample(stArg, nCycleOff, nDcNow) THEN
        _bOverflow   := TRUE;
        _nDropAppend := _nDropAppend + 1;
    END_IF

    (* Update last-value cache regardless of append success — change-detect
       should still suppress the next no-change observation. *)
    nCmpLen := _nSampleSize;
    IF nCmpLen > SIZEOF(_abyLastValue) THEN
        nCmpLen := SIZEOF(_abyLastValue);
    END_IF
    Tc2_System.MEMCPY(ADR(_abyLastValue), stArg.pValue, nCmpLen);
    _bLastValueValid := TRUE;
END_IF

_nLastSampleCycle := nNowCycle;
_bLastSampleSet   := TRUE;

(* Mid-window autoflush: when the body crosses the high-water mark we
   swap halves immediately rather than wait for _CheckFlush's push-
   interval tick. Keeps oversampling bursts streaming when one push
   window otherwise wouldn't fit.

   Critical guard — only fire when the pending half is FREE. If the
   sender is still shipping the previous frame, _DoFlush would see
   _bPending=TRUE, reset the entire active half to empty, and bump
   _nDropWindow — throwing away every sample we accumulated in the
   burst. That makes the case autoflush was designed for strictly
   worse than just letting the body hit 100 % and dropping one
   sample at a time via _nDropAppend. So: when pending is busy we
   hold off and keep filling. If we reach 100 % before pending
   drains, _AppendSample returns FALSE and we lose one sample — not
   the whole window. *)
IF _nBodyOffset >= BODY_HIGH_WATER AND NOT _bPending THEN
    _DoFlush();
END_IF

_CheckFlush();

Observe := TRUE;
END_METHOD

PROPERTY PUBLIC SampleCount : UDINT
GET
SampleCount := _nSampleCount;
END_GET
END_PROPERTY

(*
:Description: Enable / change online aggregation over the sample interval.

``nMask`` is a bitmask **OR-combined from individual ``E_MetricStat``
values**. Each set bit selects one statistic to compute via Welford
online aggregation and ship per sample tick:

==================== === ===============================================
Bit                  Hex Stat shipped per sample
==================== === ===============================================
``E_MetricStat.eMin``    1   minimum observed value
``E_MetricStat.eMax``    2   maximum observed value
``E_MetricStat.eMean``   4   arithmetic mean
``E_MetricStat.eSum``    8   sum (totalizer — energy, parts, distance)
``E_MetricStat.eCount`` 16   observations folded (gap / drop detection)
``E_MetricStat.eStdDev`` 32   standard deviation (jitter / stability)
==================== === ===============================================

The bits ship in **bit-index order** (Min first if set, then Max, Mean,
Sum, Count, StdDev). Wire size per sample = ``popcount(nMask) * 8``.

.. code-block:: pascal

	// Raw - use raw value (last), 8 B/sample (Default)
	fbEnergy.SetAggregation(0);

    // Counter — totalizer only, 8 B/sample.
    fbEnergy.SetAggregation(E_MetricStat.eSum);

    // Envelope — min + max, 16 B/sample. Catch peaks/troughs.
    fbTemp.SetAggregation(E_MetricStat.eMin OR E_MetricStat.eMax);

    // Standard — min + max + mean, 24 B/sample. Recommended default.
    fbProcess.SetAggregation(
        E_MetricStat.eMin OR E_MetricStat.eMax OR E_MetricStat.eMean);

    // Full — all six, 48 B/sample. Diagnostic / tuning.
    fbCritical.SetAggregation(
        E_MetricStat.eMin OR E_MetricStat.eMax OR E_MetricStat.eMean
        OR E_MetricStat.eSum OR E_MetricStat.eCount OR E_MetricStat.eStdDev);

Pass ``0`` to revert to raw single-value sampling. With aggregation
enabled, every ``Observe`` call updates the Welford aggregator
regardless of rate-limit; the rate-limit then controls how often the
aggregator is *snapshotted* into the body buffer. So values that
appear between sample ticks are no longer dropped — they're folded
into the next snapshot's min/max/mean/etc.

Aggregation is numeric-only. On non-numeric metrics (BOOL, STRING,
WSTRING, ENUM/discrete) the mask is ignored and a warning is logged
the first time. The mask is a hint applied at the next ``Observe``;
in-flight body content is not retroactively converted, so call
``SetAggregation`` at startup before the first ``Observe``.
*)
METHOD PUBLIC SetAggregation : BOOL
VAR_INPUT
    nMask : BYTE;
END_VAR
_nStatMask      := nMask;
_nAggSampleSize := _PopCount8(nMask) * 8;

(* If the schema is already locked to a numeric type, switch in/out of
   the aggregated body schema on the fly so the next sample tick uses
   the right write path. For non-numeric locked types the mask is held
   but never consumed (the locked schema decides which append-path runs);
   warn once so the user knows it's a no-op. *)
IF _eBodySchema = E_MetricBodySchema.eNumeric AND nMask <> 0 THEN
    _eBodySchema := E_MetricBodySchema.eNumericAggregated;
    _nSampleSize := _nAggSampleSize;
ELSIF _eBodySchema = E_MetricBodySchema.eNumericAggregated AND nMask = 0 THEN
    _eBodySchema := E_MetricBodySchema.eNumeric;
    _nSampleSize := 8;
ELSIF _eBodySchema = E_MetricBodySchema.eNumericAggregated AND nMask <> 0 THEN
    _nSampleSize := _nAggSampleSize;
ELSIF nMask <> 0 AND (_eBodySchema = E_MetricBodySchema.eBool
                   OR _eBodySchema = E_MetricBodySchema.eString
                   OR _eBodySchema = E_MetricBodySchema.eWstring
                   OR _eBodySchema = E_MetricBodySchema.eDiscrete) THEN
    F_InternalLog(
        E_LogLevel.eWarn,
        'FB_Metrics.SetAggregation',
        'Aggregation only valid for numeric metrics — %s is non-numeric, mask ignored',
        Tc2_Utilities.F_StringEx(_sName),
        Tc2_Utilities.EMPTY_ARG_VALUE,
        Tc2_Utilities.EMPTY_ARG_VALUE,
        Tc2_Utilities.EMPTY_ARG_VALUE
    );
END_IF

_AggReset();
SetAggregation := TRUE;
END_METHOD

(*
:Description: Enable / disable byte-wise change-detect (default TRUE).

Disable when you want to capture every cycle's value as-is even if it
hasn't changed (e.g. for "still alive" continuity at slow sample rates).
*)
METHOD PUBLIC SetChangeDetect : BOOL
VAR_INPUT
    bEnabled : BOOL;
END_VAR
_bChangeDetect := bEnabled;
SetChangeDetect := TRUE;
END_METHOD

(*
:Description: How often to flush the buffer to tc-otel (default 1000 ms).

Lower bound is one task cycle. Smaller values mean more frames on the wire;
larger values risk buffer overflow on high-rate metrics (8 KB ÷ sample_size).
*)
METHOD PUBLIC SetPushIntervalMs : BOOL
VAR_INPUT
    nMs : UDINT;
END_VAR
_nPushIntervalMs := nMs;
IF _nPushIntervalMs = 0 THEN
    _nPushIntervalMs := 1000;
END_IF
SetPushIntervalMs := TRUE;
END_METHOD

(*
:Description: Enable / disable per-sample timestamp emission (default FALSE).

When TRUE every body slot is prefixed with a 2-byte little-endian u16 cycle
offset relative to ``cycle_count_start``, and the wire header carries
``flags.bit2 = METRIC_FLAG_HAS_SAMPLE_TS``. Receivers use the offset to
reconstruct accurate per-sample DC times instead of linearly interpolating
across the window.

Use this when sampling is irregular — change-detect bursts, sporadic
``Observe`` calls, or `SetSampleIntervalMs` rate-limiting in combination with
bursty input. When ``Observe`` runs every task cycle, default linear
interpolation is already exact and this opt-in costs 2 B per sample for
nothing.

Side effects:

* ``_CheckFlush`` caps the push window at ``0xFFFF`` task cycles whenever
  this flag is active. On a 250 µs task that is ~16 s; on a 1 ms task
  ~65 s — well beyond any realistic metric interval. Configurations that
  would exceed the cap are silently autoflushed earlier.
* ``WithSpan`` overrides are one-shot and get consumed by the *next* flush,
  which may now be an autoflush rather than the natural window end. For
  spans that outlive one window, prefer ``BindTracer``.
* ``SetAggregation`` splits the Welford state across autoflushes, which
  produces finer-grained stat windows downstream. Acceptable for most
  dashboards; note if you rely on exact per-window moments.

Cost per sample when active: 2 B prefix. Bool (1 B) body grows to 3 B,
Numeric (8 B) to 10 B, NumericAggregated with full stat mask (48 B) to
50 B. Zero overhead when disabled.
*)
METHOD PUBLIC SetRecordSampleTimes : BOOL
VAR_INPUT
    bEnable : BOOL;
END_VAR
_bRecordSampleTimes := bEnable;
IF bEnable THEN
    (* The two sample-ts modes are mutually exclusive — the wire format
       carries them in separate flag bits but only one prefix layout per
       slot. Turning u16-offset mode on forces DC-mode off. *)
    _bRecordSampleTimesDc := FALSE;
END_IF
SetRecordSampleTimes := TRUE;
END_METHOD

(*
:Description: Enable / disable per-sample i64 absolute DC time emission (default FALSE).

Use this for **true oversampling** — when `Observe` is called more than once
per task cycle and every observation must reach the backend as its own
distinct datapoint. The u16-offset mode (``SetRecordSampleTimes``) collapses
all same-cycle samples onto one offset value; this mode emits the raw
``F_GetActualDcTime64()`` reading instead so the receiver can resolve them.

When TRUE every body slot is prefixed with an 8-byte little-endian i64
absolute DC time, and the wire header carries
``flags.bit4 = METRIC_FLAG_HAS_SAMPLE_TS_DC (0x10)``. The receiver uses
``dc_time[i]`` directly as the per-sample timestamp — no interpolation,
no dependency on ``cycle_count_*``.

**Honest timestamps, no synthetic tiebreaker**: if two consecutive
``Observe`` calls inside one task cycle happen faster than the hardware
DC clock ticks, the emitted DC times can be identical. Those duplicates
are real and may be deduplicated by storage backends with last-value-
wins semantics on identical timestamps. The PLC deliberately does *not*
fabricate a fake monotonic increment because that would lie about when
the observation actually happened.

**Mutually exclusive with ``SetRecordSampleTimes``** — calling
``SetRecordSampleTimesDc(TRUE)`` while u16-offset mode is on forces
u16-offset off, and vice versa.

**Cost** per sample when active: 8 B prefix. Bool (1 B) body grows to
9 B, Numeric (8 B) to 16 B, NumericAggregated with full stat mask
(48 B) to 56 B. Zero overhead when disabled.

**Buffer impact**: with 16 B Numeric stride the 32 KB body holds ~2048
samples per half before mid-window autoflush kicks in (at the 80 %
high-water mark). Pair with a push interval ≤ 200 ms for sustained
oversampling so the sender keeps draining between bursts.
*)
METHOD PUBLIC SetRecordSampleTimesDc : BOOL
VAR_INPUT
    bEnable : BOOL;
END_VAR
_bRecordSampleTimesDc := bEnable;
IF bEnable THEN
    _bRecordSampleTimes := FALSE;
END_IF
SetRecordSampleTimesDc := TRUE;
END_METHOD

(*
:Description: Minimum interval between captured samples (default 0 = every change).

Set > 0 to rate-limit a fast-changing value: at most one sample per ``nMs``
ms reaches the buffer, regardless of how often Observe is called.
*)
METHOD PUBLIC SetSampleIntervalMs : BOOL
VAR_INPUT
    nMs : UDINT;
END_VAR
_nSampleIntervalMs := nMs;
SetSampleIntervalMs := TRUE;
END_METHOD

(*
:Description: Override the trace-context snapshot for the very next flush.

One-shot — consumed by ``_DoFlush`` and cleared. Subsequent flushes fall
back to the ``BindTracer``-bound innermost span, or no trace at all if
neither is set.

Unlike ``BindTracer``, ``WithSpan`` captures the span **immediately**,
so it still pins the correct trace_id even if the span is ``End``'d
before flush actually runs. This is the correct tool when:

* a short-lived span closes inside the push window and you want the
  window's metrics tagged with its ID, or
* you want a specific span tagged instead of whichever happens to be
  innermost at flush time.

Typical pattern for "this metric window belongs to span X":

.. code-block:: pascal

    _spn.Begin('quick_op');
    _temp.Observe(rValue);
    _temp.WithSpan(_spn);    // pin _spn on the next flush
    _spn.End();              // span closes, but frame still carries its ID
*)
METHOD PUBLIC WithSpan : BOOL
VAR_INPUT
    pSpan : REFERENCE TO FB_Span;
END_VAR
_pSpanOverride REF= pSpan;
WithSpan := TRUE;
END_METHOD

END_FUNCTION_BLOCK

(* stored: Version 1.1.0.1, ProductVersion 3.1.4026.18
   POU FB_Metrics: Id {f4a5b6c7-d8e9-0a1b-2c3d-4e5f6a7b8c09}, SpecialFunc None
   Folder Private: Id {a5b6c7d8-e9f0-1a2b-3c4d-5e6f7a8b9c0a}
   Method _ActiveBodyPtr: Id {12345678-9abc-def0-1234-567890abcd01}
   Method _ActiveFrameAddr: Id {12345678-9abc-def0-1234-567890abcd02}
   Method _AggReset: Id {c4d5e6f7-a8b9-c0d1-e2f3-a4b5c6d7e8f0}
   Method _AggUpdate: Id {d5e6f7a8-b9c0-d1e2-f3a4-b5c6d7e8f9a0}
   Method _AnyToLreal: Id {b6c7d8e9-f0a1-2b3c-4d5e-6f7a8b9c0d0b}
   Method _AppendAggregated: Id {e6f7a8b9-c0d1-e2f3-a4b5-c6d7e8f9a0b1}
   Method _AppendSample: Id {c7d8e9f0-a1b2-3c4d-5e6f-7a8b9c0d1e0c}
   Method _CheckFlush: Id {d8e9f0a1-b2c3-4d5e-6f7a-8b9c0d1e2f0d}
   Method _DoFlush: Id {e9f0a1b2-c3d4-5e6f-7a8b-9c0d1e2f3a0e}
   Method _GetPendingLen: Id {23456789-abcd-ef01-2345-6789abcdef03}
   Method _GetPendingPtr: Id {34567890-bcde-f012-3456-789abcdef004}
   Method _LockSchema: Id {f0a1b2c3-d4e5-6f7a-8b9c-0d1e2f3a4b0f}
   Method _NotifyFrameSent: Id {45678901-cdef-0123-4567-89abcdef0005}
   Method _NowDcTime: Id {a1b2c3d4-e5f6-7a8b-9c0d-1e2f3a4b5c10}
   Method _PopCount8: Id {f7a8b9c0-d1e2-f3a4-b5c6-d7e8f9a0b1c2}
   Method BindTracer: Id {a4b5c6d7-e8f9-0011-2233-445566778899}
   Method Call: Id {b2c3d4e5-f6a7-8b9c-0d1e-2f3a4b5c6d11}
   Method FB_exit: Id {c3d4e5f6-a7b8-9c0d-1e2f-3a4b5c6d7e12}
   Method FB_Init: Id {e3a156b7-76d5-47aa-8d12-5217e8858370}
   Method Flush: Id {d4e5f6a7-b8c9-0d1e-2f3a-4b5c6d7e8f13}
   Method Init: Id {e5f6a7b8-c9d0-1e2f-3a4b-5c6d7e8f9014}
   Property MetricId: Id {f2a3b4c5-d6e7-8f90-0102-03040506071f}
   Get Get: Id {a3b4c5d6-e7f8-9001-0203-040506070820}
   Method Observe: Id {f6a7b8c9-d0e1-2f3a-4b5c-6d7e8f901015}
   Property SampleCount: Id {d0e1f2a3-b4c5-6d7e-8f90-01020304051d}
   Get Get: Id {e1f2a3b4-c5d6-7e8f-9001-02030405061e}
   Method SetAggregation: Id {a8b9c0d1-e2f3-a4b5-c6d7-e8f9a0b1c2d3}
   Method SetChangeDetect: Id {a7b8c9d0-e1f2-3a4b-5c6d-7e8f90010216}
   Method SetPushIntervalMs: Id {b8c9d0e1-f2a3-4b5c-6d7e-8f9001020317}
   Method SetRecordSampleTimes: Id {b1c2d3e4-f506-7890-a1b2-c3d4e5f60718}
   Method SetRecordSampleTimesDc: Id {c2d3e4f5-1234-5678-9abc-def012345678}
   Method SetSampleIntervalMs: Id {c9d0e1f2-a3b4-5c6d-7e8f-90010203040c}
   Method WithSpan: Id {b5c6d7e8-f9a0-1122-3344-5566778899aa} *)
